(* CoDeSys 2.3.9.47 project: OEE.pro *)
(* Libraries: STANDARD.LIB 5.6.98 11:03:02, TcBase.lib 14.5.09 11:14:08, TcSystem.lib*21.1.15 09:22:54, TcUtilities.lib*6.1.15 15:45:04 *)

(* Task configuration *)
TASK Standard (PRIORITY := 0, INTERVAL := T#1ms);
	MAIN
END_TASK

(* Global variable list: Global_Variables *)
VAR_GLOBAL

	EndMolding3 	:BOOL;
	MoldingIO 		:BOOL;

(* Vizualizacia *)
	V_Start: BOOL;
	V_Reset: BOOL;
END_VAR

(* Global variable list: Hardware *)
VAR_GLOBAL
(* Vstupy do programu *)
	Machine1  AT%I*:  ST_Machine;
	Machine2  AT%I*:  ST_Machine;
	PLCtransfer AT %I*: ARRAY[0..9] OF WORD;
(*	Errors *)
END_VAR

(* Global variable list: TwinCAT_Configuration *)
(* Generated automatically by TwinCAT - (read only) *)
VAR_CONFIG
	.Machine1 AT %IB0 : ST_Machine;
	.Machine2 AT %IB14 : ST_Machine;
	.PLCtransfer AT %IB60 : ARRAY [0..9] OF WORD;	(*  ~ {LinkedWith:TIID^Gerät 2 (CX1500-B310)^Box 1 (CX1500-B310)^10 WORD Slave-In/Master-Out^Eingänge^10 WORD Slave-In/Master-Out 8} *)
END_VAR

(* Data type *)
TYPE ST_Error_W :
STRUCT
	Byte1:BYTE;
	Byte2:BYTE;
END_STRUCT
END_TYPE

(* Data type *)
TYPE ST_Machine:
STRUCT
	STATUS 		:ST_Status;
	IO_NIO 			:ST_OK_NG;
	Error_Alarm		: ARRAY[0..15] OF ST_Error_W;
END_STRUCT
END_TYPE

(* Data type *)
TYPE ST_OK_NG :
STRUCT
	OK:BOOL;
	NG1:BOOL;
	NG2:BOOL;
	NG3:BOOL;
	NG4:BOOL;
	NG5:BOOL;
	NG6:BOOL;
	NG7:BOOL;
END_STRUCT
END_TYPE

(* Data type *)
TYPE ST_Status :
STRUCT
	MANUAL 		 : BOOL;
	SETTING 		 : BOOL;
	AUTOMATIK	 : BOOL;
	RUNING		 : BOOL;
END_STRUCT
END_TYPE

(* POU MAIN, FBD *)
PROGRAM MAIN
VAR
	fb_FILE			: FB_ADD_DATA;
	Kus				: FB_OEE;
	String1			: STRING;

	fb_FILE1			: FB_ADD_DATA;
	Kus1			: FB_OEE;
	String2			: STRING;


	Data1			: ST_OK_NG;
	Data2			: ST_OK_NG;
END_VAR
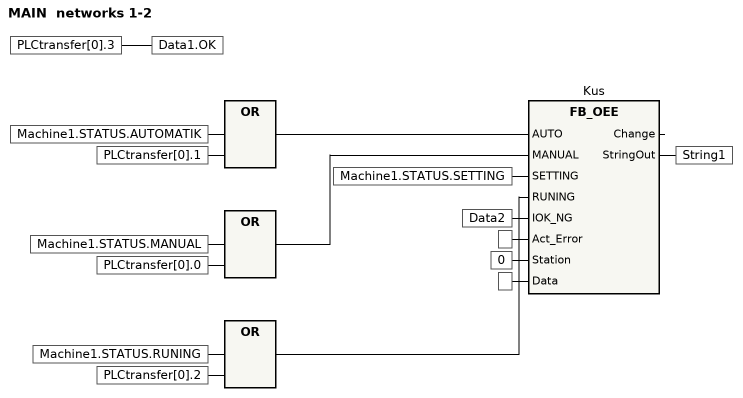
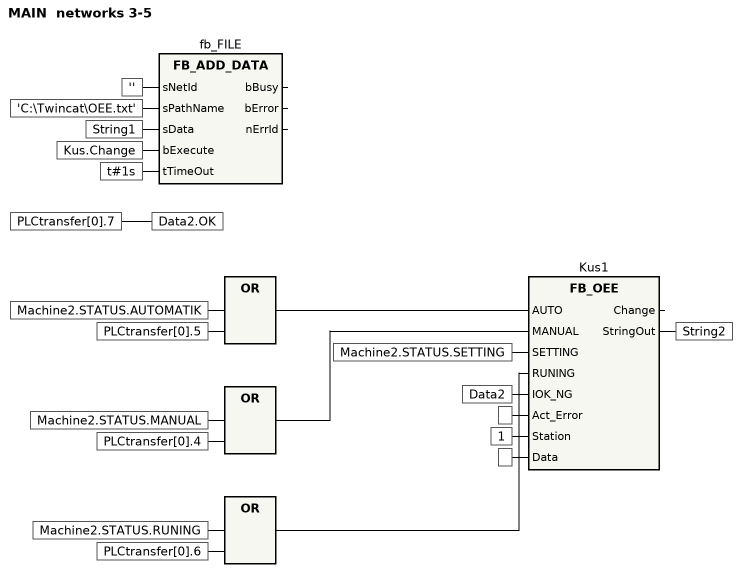
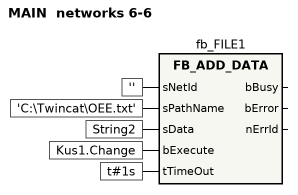
_FBD_ (* Function Block Diagram *)
NETWORK 1
	PLCtransfer[0].3 => Data1.OK
NETWORK 2
	Kus:FB_OEE(AUTO: OR(Machine1.STATUS.AUTOMATIK, PLCtransfer[0].1), MANUAL: OR(Machine1.STATUS.MANUAL, PLCtransfer[0].0), SETTING: Machine1.STATUS.SETTING, RUNING: OR(Machine1.STATUS.RUNING, PLCtransfer[0].2), IOK_NG: Data2, Act_Error: , Station: 0, Data: , StringOut => String1)
NETWORK 3
	fb_FILE:FB_ADD_DATA(sNetId: '', sPathName: 'C:\Twincat\OEE.txt', sData: String1, bExecute: Kus.Change, tTimeOut: t#1s)
NETWORK 4
	PLCtransfer[0].7 => Data2.OK
NETWORK 5
	Kus1:FB_OEE(AUTO: OR(Machine2.STATUS.AUTOMATIK, PLCtransfer[0].5), MANUAL: OR(Machine2.STATUS.MANUAL, PLCtransfer[0].4), SETTING: Machine2.STATUS.SETTING, RUNING: OR(Machine2.STATUS.RUNING, PLCtransfer[0].6), IOK_NG: Data2, Act_Error: , Station: 1, Data: , StringOut => String2)
NETWORK 6
	fb_FILE1:FB_ADD_DATA(sNetId: '', sPathName: 'C:\Twincat\OEE.txt', sData: String2, bExecute: Kus1.Change, tTimeOut: t#1s)
_END_FBD_
(* the same logic as Structured Text *)
(* Network 1 *)
Data1.OK := PLCtransfer[0].3;
(* Network 2: see the listing above *)
(* Network 3 *)
fb_FILE(sNetId := '', sPathName := 'C:\Twincat\OEE.txt', sData := String1, bExecute := Kus.Change, tTimeOut := t#1s);
(* Network 4 *)
Data2.OK := PLCtransfer[0].7;
(* Network 5: see the listing above *)
(* Network 6 *)
fb_FILE1(sNetId := '', sPathName := 'C:\Twincat\OEE.txt', sData := String2, bExecute := Kus1.Change, tTimeOut := t#1s);
END_PROGRAM

(* POU Funkcie/FB_ADD_DATA, ST *)
FUNCTION_BLOCK FB_ADD_DATA
VAR_INPUT
	sNetId			: T_AmsNetId;	(* TwinCAT sietova adresa pre cielovy subor *)
	sPathName		: T_MaxString;	(* cesta a subor pre zapis retazca *)
	sData			: STRING(150);	(* Retazec pre zapis do suboru *)
	bExecute		: BOOL; 			(* Nabezna frana odstartuje funkciu *)
	tTimeOut		: TIME := DEFAULT_ADS_TIMEOUT;(* Max. ADS timeout time *)
END_VAR
VAR_OUTPUT
	bBusy 			: BOOL;			(* TRUE => File copy execution in progress, FALSE => File copy execution idle *)
 	bError			: BOOL;			(* TRUE => Error, FALSE => No error *)
	nErrId			: UDINT;			(* Error code *)
END_VAR
VAR
	fbFileOpen		: FB_FileOpen;	(* Funkcia na otvorenie suboru *)
	fbFileClose		: FB_FileClose;	(* Funkcia na zatvorenie suboru*)
	fbFilePuts		: FB_FilePuts;		(* Funkcia prida riadok do suboru*)
	hFile			: UINT   := 0;		(* File handle of the source file *)
	Step			: DWORD;		(* Premenna pre postupnost krokov *)
	RisingEdge              : R_TRIG;		(* Nabezna hrana signalu *)
END_VAR
RisingEdge(CLK:=bExecute);

CASE Step OF
        0:      (* Cakanie na stav *)
         IF RisingEdge.Q THEN
                        bBusy := TRUE;
                        bError:= FALSE;
                        nErrId:=0;
                        Step := 1;
                        hFile:=0;
                END_IF

        1:      (* Otvor cielovy subor pre zapis *)
         fbFileOpen( bExecute := FALSE );
                fbFileOpen( sNetId := sNetId, sPathName := sPathName,
                        nMode := FOPEN_MODEAPPEND OR FOPEN_MODEPLUS,
                        ePath := PATH_GENERIC, tTimeout := tTimeOut, bExecute := TRUE );
                Step := Step + 1;
        2:       (* Kontrola otvorenia cieloveho suboru *)
                fbFileOpen( bExecute := FALSE );
                IF NOT fbFileOpen.bBusy THEN
                        IF fbFileOpen.bError THEN
                                nErrId := fbFileOpen.nErrId;
                                bError := TRUE;
                                Step := 50;
                        ELSE
                                hFile := fbFileOpen.hFile;
                                Step := Step + 1;
                        END_IF
                END_IF

        3:      (* Zapis do cieloveho suboru*)
         fbFilePuts( bExecute := FALSE );
                fbFilePuts( sNetId := sNetId, hFile:=hFile,
                        sLine := sData,
                        tTimeout := tTimeOut,
                        bExecute := TRUE );
                Step := Step+1;
        4:       (* Kontrola zapisania do suboru*)

                fbFilePuts( bExecute := FALSE );
                IF NOT fbFilePuts.bBusy THEN
                        IF fbFilePuts.bError THEN
                                nErrId := fbFilePuts.nErrId;
                                bError := TRUE;
                                Step := 50;
                        ELSE
                                Step := Step + 1;
                        END_IF
                END_IF

        5: (* Zavri cielovy subor *)
         fbFileClose( bExecute := FALSE );
                fbFileClose( sNetId:=sNetId, hFile:=hFile, bExecute:=TRUE, tTimeout:=tTimeOut );
                Step := Step + 1;
        6:
                fbFileClose( bExecute := FALSE );
                IF NOT fbFileClose.bBusy THEN
                        IF fbFileClose.bError THEN
                                nErrId := fbFileClose.nErrId;
                                bError := TRUE;
                        END_IF
                        Step := 50;
                        hFile := 0;
                END_IF

        50: (* Chyba alebo pripraveny  => vycisti *)
         IF (hFile <> 0 ) THEN
     		Step := 40; (* Zavri Cielovy subor *)
         ELSE
		 Step := 0;      (* Ready *)
		bBusy := FALSE;
         END_IF

END_CASE
END_FUNCTION_BLOCK

(* POU FB_OEE, ST *)
FUNCTION_BLOCK FB_OEE

VAR
	Status		: INT;				(* Docasne ulozenie statusu stroja *)
	Ok_NOK	: INT;				(* Docasne ulozenie vysledku kusa *)
	Temp		: STRING; 			(* Docasna premenna na ulozenie retazca *)
	sTime		: STRING;
	OKEdge			: R_TRIG;
	NG1Edge			: R_TRIG;
	NG2Edge			: R_TRIG;
	NG3Edge			: R_TRIG;
	NG4Edge			: R_TRIG;
	NG5Edge			: R_TRIG;
	NG6Edge			: R_TRIG;
	NG7Edge			: R_TRIG;

	fbTime : FB_LocalSystemTime := ( bEnable := TRUE, dwCycle := 2 );
	poc: INT;
END_VAR
VAR_INPUT
	AUTO		: BOOL := FALSE;	(* Automat zapnuty*)
	MANUAL	: BOOL := FALSE;	(* Rucne zapnute *)
	SETTING	: BOOL := FALSE;	(* Nastavovanie zapnute *)
	RUNING	: BOOL := FALSE;	(* Automatika bezi *)
 	IOK_NG 	: ST_OK_NG;		(* OK NG kus prisiel *)
	Act_Error	: INT:=0; 			(* ARRAY[0..15] OF ST_Error_W; *)
	Station		: INT:=0;			(* Cislo Stanice *)
	Data		: STRING := '';		(* Vstupne Data pred *)
END_VAR
VAR_OUTPUT
	Change		: BOOL;				(* Signal pre start zapisu *)
	StringOut	: STRING;			(* Vystupny retazec pre zapis *)
END_VAR
VAR PERSISTENT
	stemp		: INT ;				(* Pamet predchadzajuceho stavu status *)
	Old_Error	: INT;				(* ARRAY[0..15] OF ST_Error_W;*)
END_VAR
(* Ziskanie aktualneho casu zo systemu.*)

fbTime();
sTime :=   SYSTEMTIME_TO_STRING(fbTime.systemTime);

(*Data:= CONCAT (sTime,'|');   (*Doplnenie oddelovaca *)

(* Reset premennych.*)
Change:=0;			(*Zmena stavu *)
Status:= 0;
Ok_NOK:=-1;		(*Stav -1 je rozpracovany kus alebo bola iba zmena stavu stroja*)

(* Zistenie stavu stroja Auto Manual ..*)
IF RUNING		THEN Status:= 8 ; END_IF;
IF AUTO		AND Status<4	 THEN Status:= 4 ; END_IF;
IF SETTING  	AND Status<2	 THEN Status:= 2 ; END_IF;
IF MANUAL		AND Status<1	 THEN Status:= 1 ; END_IF;

(*Zistenie nabeznej hrany signalov od kusa*)
OKEdge(CLK:=IOK_NG.OK);
NG1Edge(CLK:=IOK_NG.NG1);
NG2Edge(CLK:=IOK_NG.NG2);
NG3Edge(CLK:=IOK_NG.NG3);
NG4Edge(CLK:=IOK_NG.NG4);
NG5Edge(CLK:=IOK_NG.NG5);
NG6Edge(CLK:=IOK_NG.NG6);
NG7Edge(CLK:=IOK_NG.NG7);

(* Zistenie vyrobeneho kusa OK/NG a zapisanie hodnoty do Ok_NOK*)
IF OKEdge.Q THEN Ok_NOK:=0; END_IF;
IF NG1Edge.Q THEN Ok_NOK:=1; END_IF;
IF NG2Edge.Q THEN Ok_NOK:=2; END_IF;
IF NG3Edge.Q THEN Ok_NOK:=3; END_IF;
IF NG4Edge.Q THEN Ok_NOK:=4; END_IF;
IF NG5Edge.Q THEN Ok_NOK:=5; END_IF;
IF NG6Edge.Q THEN Ok_NOK:=6; END_IF;
IF NG7Edge.Q THEN Ok_NOK:=7; END_IF;

(* Osetrenie poslania stavu pri starte twincatu *)
IF  fbTime.systemTime.wYear = 1970 THEN
	Stemp:=Status;
END_IF;

(* Zistenie zmeny na Statuse a OK_NG*)
IF (Status  <> stemp OR Ok_NOK >= 0 OR Act_Error <> Old_Error)  AND fbTime.systemTime.wYear<>1970THEN
Stemp:=Status;	(**)

Change:=1;		(*bola zistena zmena na STATUS alebo na OK_NOK*)
END_IF;

(* Zapisanie vysledku po zisteni zmeny  *)

IF Change  THEN

(* FOR poc:=0 TO 15 DO 1*)
	Data:= CONCAT (sTime,'|');			(* Cas *)
	Temp:=INT_TO_STRING(Station);	(*Cislo stanice*)
	Data:=CONCAT(Data,Temp);
	Data:=CONCAT(Data,'|');
	Temp:=INT_TO_STRING(Status);	(*Status stroja*)
	Data:=CONCAT(Data,Temp);
	Data:=CONCAT(Data,'|');
	Temp:=INT_TO_STRING(Ok_NOK);	(*OK_NOK*)
	Data:=CONCAT(Data,Temp);
	Data:=CONCAT(Data,'|');
	Temp:=INT_TO_STRING(Act_Error);	(*Aktual_Error*)
	Data:=CONCAT(Data,Temp);
	Data:=CONCAT(Data,'|');
	Temp:=INT_TO_STRING(Old_Error);	(*Old_Error*)
	Data:=CONCAT(Data,Temp);
	Data:=CONCAT(Data,'|');
	StringOut:=CONCAT(Data,' $L');		(*New Line*)





(* Old_Error:= Act_Error; *)
END_IF;

(*TP1(IN:= Change, PT:=t#3s , Q=>Change , ET=> );*)
END_FUNCTION_BLOCK

(* Visualisation START
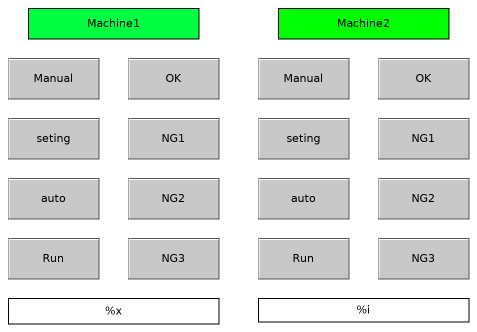
button at (30,250)-(121,291): text "auto"; toggles Machine1.STATUS.AUTOMATIK
button at (30,130)-(121,171): text "Manual"; toggles Machine1.STATUS.MANUAL
button at (30,190)-(121,231): text "seting"; toggles Machine1.STATUS.SETTING
button at (30,310)-(121,351): text "Run"; toggles Machine1.STATUS.RUNING
rectangle at (30,370)-(241,396): text "%x"; shows Machine1.Error_Alarm; editable
button at (150,130)-(241,171): text "OK"; taps Machine1.IO_NIO.OK
button at (150,190)-(241,231): text "NG1"; taps Machine1.IO_NIO.NG1
button at (150,250)-(241,291): text "NG2"; taps Machine1.IO_NIO.NG2
button at (150,310)-(241,351): text "NG3"; taps Machine1.IO_NIO.NG3
button at (280,250)-(371,291): text "auto"; toggles Machine2.STATUS.AUTOMATIK
button at (280,130)-(371,171): text "Manual"; toggles Machine2.STATUS.MANUAL
button at (280,190)-(371,231): text "seting"; toggles Machine2.STATUS.SETTING
button at (280,310)-(371,351): text "Run"; toggles Machine2.STATUS.RUNING
button at (400,130)-(491,171): text "OK"; taps Machine2.IO_NIO.OK
button at (400,190)-(491,231): text "NG1"; taps Machine2.IO_NIO.NG1
button at (400,250)-(491,291): text "NG2"; taps Machine2.IO_NIO.NG2
button at (400,310)-(491,351): text "NG3"; taps Machine2.IO_NIO.NG3
rectangle at (280,370)-(491,394): text "%i"; shows MAIN.Test
rectangle at (50,80)-(221,111): text "Machine1"
rectangle at (300,80)-(471,111): text "Machine2"
*)
